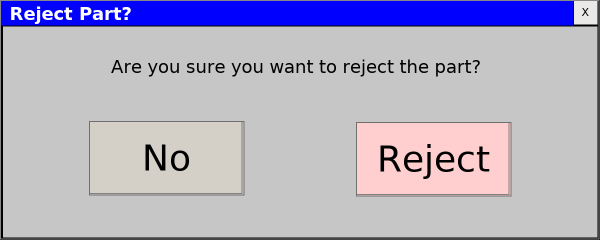
VISUALIZATION dialogReject  // 600x240
    Rectangle (0,0 600x240)
    Button (356,122 155x74), "Reject"
        OnMouseClick: CloseDialog Dialog=dialogReject, Result=Yes, NumpadKeypadSet=True
    Button (89,121 155x74), "No"
        OnMouseClick: CloseDialog Dialog=dialogReject, Result=No, NumpadKeypadSet=True
    Label (74,43 444x48), "Are you sure you want to reject the part?"
    Rectangle (0,0 600x26), "Reject Part?"
    Rectangle (573,0 25x25), "X"
        OnMouseClick: CloseDialog Dialog=dialogReject, Result=Cancel, NumpadKeypadSet=True
END_VISUALIZATION

(* stored: Version 1.1.0.1, ProductVersion 3.1.4024.12
   Visu dialogReject: Id {60b73fab-2b7e-49e9-929e-bc324a4c45f0} *)
